// TwinCAT 3 PLC project PLC
// ProgramVersion: 3.1.4026.20
// CompilerDefines: VISU_USEPROPERTYINFO
// libraries:
//   SPT Base Types, * (Beckhoff Automation LLC)
//   SPT Components, * (Beckhoff Automation LLC)
//   SPT Diagnostic, * (Beckhoff Automation LLC)
//   SPT EtherCat, * (Beckhoff Automation LLC)
//   SPT Event Logger, * (Beckhoff Automation LLC)
//   SPT Motion Control, * (Beckhoff Automation LLC)
//   SPT Utilities, * (Beckhoff Automation LLC)
//   SPT Vision, * (Beckhoff Automation LLC)
//   Tc2_MC2, * (Beckhoff Automation GmbH)
//   Tc2_MC2_Camming, * (Beckhoff Automation GmbH)
//   Tc2_Standard, * (Beckhoff Automation GmbH)
//   Tc2_System, * (Beckhoff Automation GmbH)
//   Tc3_EventLogger, * (Beckhoff Automation GmbH)
//   Tc3_MC2_AdvancedHoming, * (Beckhoff Automation GmbH)
//   Tc3_McCollisionAvoidance, * (Beckhoff Automation GmbH)
//   Tc3_McCoordinatedMotion, * (Beckhoff Automation GmbH)
//   Tc3_PackML_V3, * (Beckhoff Automation GmbH)
//   Tc3_Vision, * (Beckhoff Automation GmbH)
// project tree:
//   / GlobalTextList.TcGTLO (not stored), PlcTask.TcTTO (not stored), VisionTask.TcTTO, VisualizationManager.TcVMO (not stored)
//   POUs/ FB_VisionController.TcPOU, Machine.TcPOU, MAIN.TcPOU (not stored), Vision.TcPOU (not stored)
//   POUs/EquipmentModules/ FB_VisionOrientation.TcPOU (not stored)
//   VISUs/ Visualization.TcVIS
// real-time tasks:
//   TASK PlcTask: cycle T#100000us, priority 20, ADS port 350
//   TASK Job Task: cycle default, priority 32
//   TASK VnTask ImgAcq (Camera1): cycle T#1ms, priority 5, ADS port 351
//   TASK VnTask ADS (Camera1): cycle T#10ms, priority 6, ADS port 352
//   TASK VisionTask: cycle T#1ms, priority 21, ADS port 353
// motion (NC):
//   TASK NC-Task 1 SAF: cycle T#2ms, priority 4, ADS port 501
//   TASK NC-Task 1 SVB: cycle T#10ms, priority 8, ADS port 511
//   AXIS CanRotation (id 2)
//     General: UnitName=°, UnitFlags=#x00000004
//     Dynamic: Acceleration=3214.611, Deceleration=3214.611, Jerk=9643.833
//     Velo: RefSearch=21.43074, RefSync=21.43074, SlowManual=107.1537, FastManual=642.9222, Fast=2143.074, Maximum=2143.074
//     OtherSettings: AllowMotionCmdToSlave=true
//     encoder EncType=19
//       EncPara: ScaleFactorNumerator=360, ScaleFactorDenominator=1048576, MaxCount=#xffffffff
//     drive DrvType=16
//       DrvPara: MaxCount=#xffffffff, DriveControlDWord=#x00020100
//         Analog: VeloReferenz=2357.3814, VeloScale=32, TorqueSetpointScale=10, ScaleFactorActTorque=0.1
//         TimeComp: TaskDelayCycles=1
//     controller CtrType=1
//       CtrPara: PriorControlFactor=1
//         Observer: BandWidth=20
// I/O:
//   DEVICE Device 2 (EtherCAT), AmsNetId 192.168.1.213.3.1
//     Term 4 (EK1818) [EK1818 EtherCAT IO-Coupler  (1A E-Bus, 8 Ch. Dig. In, 3ms, 4 Ch. Dig. Out 24V, 0,5A)]
//       Term 5 (ELM7212-0010) [ELM7212-0010 2Ch. Servo Terminal (48 V, 4,5 A RMS, OCT)]
//       Term 6 (EK1310) [EK1310 EtherCAT P extension with feed-in]
//     Box 7 (VCS2000-0200) [VCS2000-0200 | Area scan camera, 2.5 GBit/s, Sony IMX392, monochrome, 2.3 MP]
//       modules: Device, GenICam
//   DEVICE Device 1 (RT-Ethernet Adapter)
// variable links:
//   NC-Task 1 SAF/Axes/CanRotation <-> Device 2 (EtherCAT)/Term 4 (EK1818)/Term 5 (ELM7212-0010)
//     Drive/Inputs/In/nDataIn1 <-> DRV Following error actual value Channel 1/Following error actual value
//     Drive/Inputs/In/nDcOutputTime <-> InfoData/DcOutputShift
//     Drive/Inputs/In/nState1 <-> DRV Statusword Channel 1/Statusword
//     Drive/Inputs/In/nState2 <-> DRV Statusword Channel 1/Statusword @bit 8
//     Drive/Inputs/In/nState4 @bit 1 <-> WcState/InputToggle
//     Drive/Inputs/In/nState4 <-> WcState/WcState
//     Drive/Outputs/Out/nCtrl1 <-> DRV Controlword Channel 1/Controlword
//     Drive/Outputs/Out/nCtrl2 <-> DRV Controlword Channel 1/Controlword @bit 8
//     Drive/Outputs/Out/nDataOut1 <-> DRV Target position Channel 1/Target position
//     Enc/Inputs/In/nDataIn1 <-> FB Position Channel 1/Position
//     Enc/Inputs/In/nDcInputTime <-> InfoData/DcInputShift
//     Enc/Inputs/In/nState4 @bit 1 <-> WcState/InputToggle
//     Enc/Inputs/In/nState4 <-> WcState/WcState
//   PLC/PLC Instance <-> NC-Task 1 SAF/Axes/CanRotation
//     PlcTask Inputs/MAIN.Machine.VisionOrientation.SpinAxis.BasicAxis._Axis.NcToPlc <-> Outputs/ToPlc
//     PlcTask Outputs/MAIN.Machine.VisionOrientation.SpinAxis.BasicAxis._Axis.PlcToNc <-> Inputs/FromPlc
//   PLC/PLC Instance <-> PLC/PLC Instance
//     PlcTask Inputs/MAIN.Machine.VisionOrientation.Camera.CameraState <-> VisionTask Outputs/Vision.VisionBase.CameraState
//     PlcTask Inputs/MAIN.Machine.VisionOrientation.Camera.NumberOfResults <-> VisionTask Outputs/Vision.VisionBase.NumberOfResults
//     PlcTask Inputs/MAIN.Machine.VisionOrientation.Camera.Results <-> VisionTask Outputs/Vision.VisionBase.Results
//     PlcTask Inputs/MAIN.Machine.VisionOrientation.Camera.ResultsAvailable <-> VisionTask Outputs/Vision.VisionBase.ResultsAvailable
//     PlcTask Inputs/MAIN.Machine.VisionOrientation.Camera.VisionError <-> VisionTask Outputs/Vision.VisionBase.VisionError
//     PlcTask Inputs/MAIN.Machine.VisionOrientation.Camera.VisionErrorID <-> VisionTask Outputs/Vision.VisionBase.VisionErrorID
//     VisionTask Inputs/Vision.VisionBase.Reset <-> PlcTask Outputs/MAIN.Machine.VisionOrientation.Camera._Reset
//     VisionTask Inputs/Vision.VisionBase.ResultsReceived <-> PlcTask Outputs/MAIN.Machine.VisionOrientation.Camera.ResultsReceived
//     VisionTask Inputs/Vision.VisionBase.RunVision <-> PlcTask Outputs/MAIN.Machine.VisionOrientation.Camera._RunVision
//     VisionTask Inputs/Vision.VisionBase.SoftwareTrigger <-> PlcTask Outputs/MAIN.Machine.VisionOrientation.Camera.SoftwareTrigger

CONFIGURATION PLC
    RESOURCE PLC ON TwinCAT3
        TASK VisionTask(INTERVAL := T#1ms, PRIORITY := 21);
        PROGRAM Vision WITH VisionTask : Vision;
    END_RESOURCE
END_CONFIGURATION

// ---- POUs/FB_VisionController.TcPOU
FUNCTION_BLOCK FB_VisionController EXTENDS FB_VisionCameraBase
VAR_INPUT
END_VAR
VAR_OUTPUT
END_VAR
VAR
END_VAR

METHOD ProcessImage
END_METHOD

END_FUNCTION_BLOCK

// ---- POUs/Machine.TcPOU
FUNCTION_BLOCK Machine EXTENDS FB_PackML_BaseModule
VAR
	VisionOrientation	: FB_VisionOrientation;
END_VAR

METHOD PROTECTED HMIPermissions
AllowHMIControl(TRUE);
END_METHOD

(* Basic module initialization logic*)
METHOD PROTECTED Initialize : BOOL
Initialize := FALSE;
CASE DescendantSequenceState OF
	0:
		RegisterSubmodule(SubModule := VisionOrientation);
		DescendantSequenceState := DescendantSequenceState + 10;

	10:
		IF SUPER^.Initialize() THEN
			Initialize := TRUE;
		END_IF
END_CASE
END_METHOD

END_FUNCTION_BLOCK

// ---- VISUs/Visualization.TcVIS
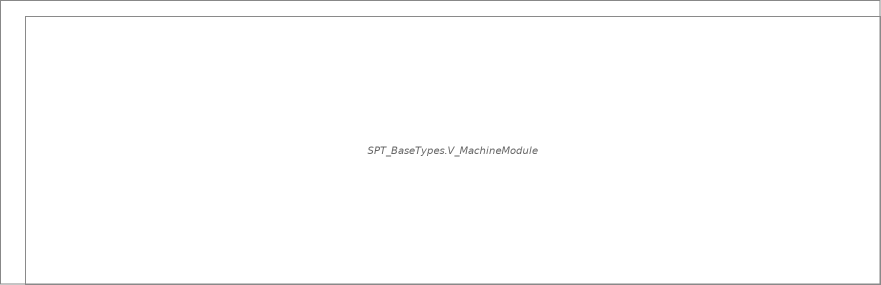
VISUALIZATION Visualization  // 881x285
    Frame (25,16 856x269)
        shows SPT_BaseTypes.V_MachineModule(HMI := MAIN.Machine.PackMLBaseModule_HMI)
END_VISUALIZATION
